(* CODESYS project FB_TESTING.PleaseIhaveKids.xml

Project tree, tasks and I/O mapping:
*)

// PleaseIhaveKids
ACTION PleaseIhaveKids:
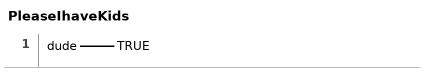
// NETWORK 1
TRUE := dude;
END_ACTION
